Universal Robots PolyScope program: hookB_manager.urp

Program hookB_manager (installation=admin directory=/programs/THU_530PM createdIn=3.15.8.106339 lastSavedIn=3.15.8.106339 robotSerialNumber=2015350926)
Calibrated DH parameters: a=[0, -0.425, -0.39225, 0, 0, 0]; d=[0.089159, 0, 0, 0.10915, 0.09465, 0.0823]; alpha=[1.570796, 0, 0, 1.570796, -1.570796, 0]; deltaTheta=[0, 0, 0, 0, 0, 0]
Robot Program (runOnlyOnce=true)
  above_HookB := p[-0.39636, -0.32475, 0.15692, 2.226, -2.216, 0.000]
  offset_x := hook_indexB * 0.047
  above_pose_B := pose_add(above_HookB, p[0.0, -offset_x, 0.0, 0.0, 0.0, 0.0])
  at_pose_B := pose_add(above_pose_B, p[0.0, 0.0, -0.10503, 0.0, 0.0, 0.0])
  Script: movel (get_inverse_kin(above_pose_B))
  Script: movel (get_inverse_kin(at_pose_B))
  Set DigitalOutput pin=digital_out[0]; digitalValue=1
  Wait Sleep waitTime=1
  Script: movel (get_inverse_kin(above_pose_B), a = 0.5, v = 0.1)
  Script: movej (get_inverse_kin(above_HookB))
  hook_indexB := hook_indexB + 1
  If hook_index ≥ num_hooks
    hook_indexB := 0
    Popup Message (haltProgram=false message=All Hook_B's were used! Reload Fixture inputType=Text)
